// TwinCAT 3 PLC project Untitled1
// ProgramVersion: 3.1.4024.0
// libraries:
//   Tc2_MC2, * (Beckhoff Automation GmbH)
//   Tc2_MC2_Drive, * (Beckhoff Automation GmbH)
//   Tc2_Standard, * (Beckhoff Automation GmbH)
//   Tc2_System, * (Beckhoff Automation GmbH)
//   Tc3_Module, * (Beckhoff Automation GmbH)
// project tree:
//   GVLs/ GVL.TcGVL
//   / PlcTask.TcTTO
//   POUs/ Get_PID_Gain.TcPOU, Init.TcPOU, MAIN.TcPOU
// real-time tasks:
//   TASK PlcTask: cycle T#10ms, priority 20, ADS port 350
// motion (NC):
//   TASK NC-Task 1 SAF: cycle T#2ms, priority 4, ADS port 501
//   TASK NC-Task 1 SVB: cycle T#10ms, priority 8, ADS port 511
//   AXIS Axis 1 (id 1)
//     OtherSettings: AllowMotionCmdToSlave=true
//     encoder EncType=19
//       EncPara: MaxCount=#xffffffff
//     drive DrvType=16
//       DrvPara: MaxCount=#xffffffff, DriveControlDWord=#x00020100
//         Analog: TorqueSetpointScale=10, ScaleFactorActTorque=0.1
//         TimeComp: TaskDelayCycles=1
//     controller CtrType=1
//       CtrPara: PriorControlFactor=1
//         PosDiffControl: Enable=false
//         Observer: BandWidth=20
//   AXIS Axis 2 (id 2)
//     OtherSettings: AllowMotionCmdToSlave=true
//     encoder EncType=19
//       EncPara: MaxCount=#xffffffff
//     drive DrvType=16
//       DrvPara: MaxCount=#xffffffff, DriveControlDWord=#x00020100
//         Analog: TorqueSetpointScale=10, ScaleFactorActTorque=0.1
//         TimeComp: TaskDelayCycles=1
//     controller CtrType=1
//       CtrPara: PriorControlFactor=1
//         PosDiffControl: Enable=false
//         Observer: BandWidth=20
// I/O:
//   DEVICE Device 3 (EtherCAT), AmsNetId 169.254.80.96.4.1
//     Drive 1 (MADHT1505BA1) [MADHT1505BA1]
//     Drive 2 (MADHT1507BA1) [MADHT1507BA1]
// variable links:
//   NC-Task 1 SAF/Axes/Axis 1 <-> Device 3 (EtherCAT)/Drive 1 (MADHT1505BA1)
//     Drive/Inputs/In/nDataIn1 <-> Transmit PDO mapping 1/Following error actual value
//     Drive/Inputs/In/nState1 <-> Transmit PDO mapping 1/Statusword
//     Drive/Inputs/In/nState2 <-> Transmit PDO mapping 1/Statusword @bit 8
//     Drive/Inputs/In/nState4 @bit 1 <-> WcState/InputToggle
//     Drive/Inputs/In/nState4 <-> WcState/WcState
//     Drive/Inputs/In/nState5 <-> Transmit PDO mapping 1/Modes of operation display
//     Drive/Outputs/Out/nCtrl1 <-> Receive PDO mapping 1/Controlword
//     Drive/Outputs/Out/nCtrl2 <-> Receive PDO mapping 1/Controlword @bit 8
//     Drive/Outputs/Out/nCtrl5 <-> Receive PDO mapping 1/Modes of operation
//     Drive/Outputs/Out/nDataOut1 <-> Receive PDO mapping 1/Target position
//     Enc/Inputs/In/nDataIn1 <-> Transmit PDO mapping 1/Position actual value
//     Enc/Inputs/In/nDataIn3 <-> Transmit PDO mapping 1/Touch probe pos1 pos value
//     Enc/Inputs/In/nState4 @bit 1 <-> WcState/InputToggle
//     Enc/Inputs/In/nState4 <-> WcState/WcState
//     Enc/Inputs/In/nState5 <-> Transmit PDO mapping 1/Touch probe status
//     Enc/Inputs/In/nState6 <-> Transmit PDO mapping 1/Touch probe status @bit 8
//     Enc/Outputs/Out/nCtrl5 <-> Receive PDO mapping 1/Touch probe function
//     Enc/Outputs/Out/nCtrl6 <-> Receive PDO mapping 1/Touch probe function @bit 8
//   NC-Task 1 SAF/Axes/Axis 2 <-> Device 3 (EtherCAT)/Drive 2 (MADHT1507BA1)
//     Drive/Inputs/In/nDataIn1 <-> Transmit PDO mapping 1/Following error actual value
//     Drive/Inputs/In/nState1 <-> Transmit PDO mapping 1/Statusword
//     Drive/Inputs/In/nState2 <-> Transmit PDO mapping 1/Statusword @bit 8
//     Drive/Inputs/In/nState4 @bit 1 <-> WcState/InputToggle
//     Drive/Inputs/In/nState4 <-> WcState/WcState
//     Drive/Inputs/In/nState5 <-> Transmit PDO mapping 1/Modes of operation display
//     Drive/Outputs/Out/nCtrl1 <-> Receive PDO mapping 1/Controlword
//     Drive/Outputs/Out/nCtrl2 <-> Receive PDO mapping 1/Controlword @bit 8
//     Drive/Outputs/Out/nCtrl5 <-> Receive PDO mapping 1/Modes of operation
//     Drive/Outputs/Out/nDataOut1 <-> Receive PDO mapping 1/Target position
//     Enc/Inputs/In/nDataIn1 <-> Transmit PDO mapping 1/Position actual value
//     Enc/Inputs/In/nDataIn3 <-> Transmit PDO mapping 1/Touch probe pos1 pos value
//     Enc/Inputs/In/nState4 @bit 1 <-> WcState/InputToggle
//     Enc/Inputs/In/nState4 <-> WcState/WcState
//     Enc/Inputs/In/nState5 <-> Transmit PDO mapping 1/Touch probe status
//     Enc/Inputs/In/nState6 <-> Transmit PDO mapping 1/Touch probe status @bit 8
//     Enc/Outputs/Out/nCtrl5 <-> Receive PDO mapping 1/Touch probe function
//     Enc/Outputs/Out/nCtrl6 <-> Receive PDO mapping 1/Touch probe function @bit 8
//   Untitled1/Untitled1 Instance <-> NC-Task 1 SAF/Axes/Axis 1
//     PlcTask Inputs/GVL.AxisY.NcToPlc <-> Outputs/ToPlc
//     PlcTask Outputs/GVL.AxisY.PlcToNc <-> Inputs/FromPlc
//   Untitled1/Untitled1 Instance <-> NC-Task 1 SAF/Axes/Axis 2
//     PlcTask Inputs/GVL.AxisX.NcToPlc <-> Outputs/ToPlc
//     PlcTask Outputs/GVL.AxisX.PlcToNc <-> Inputs/FromPlc

CONFIGURATION Untitled1
    RESOURCE PLC ON TwinCAT3
        TASK PlcTask(INTERVAL := T#10ms, PRIORITY := 20);
        PROGRAM MAIN WITH PlcTask : MAIN;
    END_RESOURCE
END_CONFIGURATION

// ---- GVLs/GVL.TcGVL
{attribute 'qualified_only'}
VAR_GLOBAL
			AxisX : AXIS_REF;
			AxisY : AXIS_REF;
			
			//Moter Power	
			AxisX_Power_Fuc : MC_Power;
			AxisY_Power_Fuc : MC_Power;
					
			OnMoterX : BOOL;
			OnMoterY : BOOL;
			
			//***************Stop***********//
			X_Stop : MC_Stop;
			X_Stop_EX :BOOL :=FALSE;
			Y_Stop : MC_Stop;
			Y_Stop_EX :BOOL :=FALSE;
			//**************Jog***********//
			
			X_Jog : MC_Jog;
			Y_Jog : MC_Jog;
			X_FW : BOOL :=FALSE;
			X_BW : BOOL :=FALSE;
			//**************Pos_Offset_Clear***********//
			
			X_Pos_Offset_EX  : BOOL :=FALSE;
			Y_Pos_Offset_EX : BOOL :=FALSE;
			
			
			//***************Moter Move***************//
			AxisX_AbMove_Fuc :MC_MoveAbsolute;
			AxisY_AbMove_Fuc :MC_MoveAbsolute;
			
			//Moter GetVelocity
			X_GetVel: MC_ReadActualVelocity;
   			Y_GetVel: MC_ReadActualVelocity;
			X_Vel  : LREAL;
			Y_Vel  : LREAL;	
			
			//Moter GetPosition
			X_GetPos :MC_ReadActualPosition;
			Y_GetPos :MC_ReadActualPosition;
	  		X_Pos : LREAL;	  	  
	  		Y_Pos : LREAL;
			
			//Input
			X_Command_Vel : LREAL := 200;     
			X_Command_Acc : LREAL :=200;
			X_Command_Dec : LREAL :=200;
			X_AbMove_Ex : BOOL := FALSE;
			X_Command_Pos : LREAL :=0;
			
			Y_Command_Vel : LREAL := 200;     
			Y_Command_Acc : LREAL := 200;
			Y_Command_Dec : LREAL := 200;
			Y_AbMove_Ex : BOOL := FALSE;
			Y_Command_Pos : LREAL := 0;
			
				
			//Output
			X_Busy : BOOL;
			Y_Busy : BOOL;
			
			X_Error :BOOL;
			Y_Error :BOOL;
			
			X_ErrorID :UDINT;
			Y_ErrorID :UDINT;
			
			X_Done : BOOL;
			Y_Done : BOOL;	
		 //***************Moter Move End***************//
			
		//PID 
			
       		 fbCoEReadP_X:FB_CoERead;
			fbCoEReadI_X:FB_CoERead;
			fbCoEReadD_X:FB_CoERead;
			
			fbCoEReadP_Y:FB_CoERead;
			fbCoEReadI_Y:FB_CoERead;
			fbCoEReadD_Y:FB_CoERead;
			
			fbCoERead_Y:FB_CoERead;
			
			Index: WORD :=16#3100; 
			X_Gain: WORD :=400 ;
			Y_Gain: WORD :=400 ;
			X_COE_Ex :BOOL :=FALSE;
			Y_COE_Ex :BOOL :=FALSE;
			CompleteAccess: BOOL := FALSE; 
   			Success: BOOL; 
			
			X_GetP_Gain : WORD;
			X_GetI_Gain : WORD;
			X_GetD_Gain : WORD;
			X_CoERead_EX  :BOOL:=TRUE;
			
			Y_GetP_Gain : WORD;
			Y_GetI_Gain : WORD;
			Y_GetD_Gain : WORD;
			Y_CoERead_EX  :BOOL:=TRUE;
			//PID End
END_VAR

// ---- POUs/MAIN.TcPOU
PROGRAM MAIN
VAR
		Y_SetZero_Func: MC_SetPosition;
	
	    X_SetZero_Func: MC_SetPosition;
END_VAR


Y_SetZero_Func.Options.ClearPositionOffset :=TRUE;
Y_SetZero_Func(
		Axis :=GVL.AxisX,
		Position := ,
		Execute := GVL.X_Pos_Offset_EX,
);

X_SetZero_Func.Options.ClearPositionOffset :=TRUE;
X_SetZero_Func(
		Axis :=GVL.AxisY,
		Position := ,
		Execute := GVL.Y_Pos_Offset_EX,
);


Init();
Get_PID_Gain();


GVL.AxisX_Power_Fuc.Enable := GVL.OnMoterX;
GVL.AxisY_Power_Fuc.Enable := GVL.OnMoterY;



GVL.AxisX_AbMove_Fuc.Execute := GVL.X_AbMove_Ex;

IF NOT GVL.X_Busy THEN	
	GVL.X_AbMove_Ex := FALSE;
END_IF



GVL.AxisY_AbMove_Fuc.Execute := GVL.Y_AbMove_Ex;
IF NOT GVL.Y_Busy THEN	
	GVL.Y_AbMove_Ex := FALSE;
END_IF

END_PROGRAM

// ---- POUs/Init.TcPOU
FUNCTION Init : BOOL
VAR_INPUT
END_VAR
VAR
	IsComplete : BOOL;
END_VAR


GVL.X_Stop(
	 Axis := GVL.AxisX,
	 Execute :=GVL.X_Stop_EX
);

GVL.Y_Stop(
	 Axis := GVL.AxisY,
	 Execute :=GVL.Y_Stop_EX
);

GVL.X_Jog(

    Axis := GVL.AxisX,

    JogForward := GVL.X_FW,

    JogBackwards := GVL.X_BW,

    Position := 50,

    Velocity := 500,

    Mode := E_JogMode.MC_JOGMODE_INCHING
);



GVL.AxisX_Power_Fuc(
			Axis := GVL.AxisX,
			Enable_Negative :=TRUE,
			Enable_Positive := TRUE,
			Override := 100,
			Enable :=GVL.OnMoterX
			);	
			
GVL.AxisY_Power_Fuc(
			Axis := GVL.AxisY,
			Enable_Negative :=TRUE,
			Enable_Positive := TRUE,
			Override := 100,
			Enable :=GVL.OnMoterY
			);	
			
GVL.AxisX_AbMove_Fuc(
	Axis := GVL.AxisX,
	Acceleration := GVL.X_Command_Acc,
	Velocity := GVL.X_Command_Vel,
	Deceleration := GVL.X_Command_Dec,
	Position :=GVL.X_Command_Pos,
	Busy => GVL.X_Busy,
	Done => GVL.X_Done
	);
	
GVL.AxisY_AbMove_Fuc(
	Axis := GVL.AxisY,
	Acceleration := GVL.Y_Command_Acc,
	Velocity := GVL.Y_Command_Vel,
	Deceleration := GVL.Y_Command_Dec,
	Position :=GVL.Y_Command_Pos,
	Busy => GVL.Y_Busy,
	Error => GVL.Y_Error,
	ErrorID => GVL.Y_ErrorID,
	);
	
// Get Velocity and Position for PID Graph // 
GVL.X_GetVel(
	Axis :=GVL.AxisX,
	Enable := TRUE,
	ActualVelocity =>GVL.X_Vel
	);
GVL.Y_GetVel(
	Axis :=GVL.AxisY,
	Enable := TRUE,
	ActualVelocity =>GVL.Y_Vel
	);
GVL.X_GetPos(
	Axis := GVL.AxisX,
	Enable := TRUE,
	Position => GVL.X_Pos,
	);
GVL.Y_GetPos(
	Axis := GVL.AxisY,
	Enable := TRUE,
	Position => GVL.Y_Pos,
	);

END_FUNCTION

// ---- POUs/Get_PID_Gain.TcPOU
FUNCTION Get_PID_Gain : bool
VAR_INPUT
END_VAR
VAR
END_VAR

GVL.fbCoEReadP_X(
		Axis :=GVL.AxisX,		
		NetId := '169.254.80.96.1.1',   //target NetID 
  		Index := 16#3100,
  		pDstBuf := ADR(GVL.X_GetP_Gain), 
  		BufLen := SIZEOF(GVL.X_GetP_Gain), 
  		Execute := GVL.X_CoERead_EX, 
  		Timeout := T#1S, 	
	);	
GVL.fbCoEReadD_X(
		Axis :=GVL.AxisX,		
		NetId := '169.254.80.96.1.1', 
  		Index := 16#3101,
  		pDstBuf := ADR(GVL.X_GetD_Gain), 
  		BufLen := SIZEOF(GVL.X_GetD_Gain), 
  		Execute := GVL.X_CoERead_EX, 
  		Timeout := T#1S, 	
		
	);	
GVL.fbCoEReadI_X(
		Axis :=GVL.AxisX,		
		NetId := '169.254.80.96.1.1', 
  		Index := 16#3102,
  		pDstBuf := ADR(GVL.X_GetI_Gain), 
  		BufLen := SIZEOF(GVL.X_GetI_Gain), 
  		Execute := GVL.X_CoERead_EX, 
  		Timeout := T#1S, 	
	);	
GVL.X_CoERead_EX := FALSE;
	
GVL.fbCoEReadP_Y(
		Axis :=GVL.AxisY,		
		NetId := '169.254.80.96.1.1', 
  		Index := 16#3100,
  		pDstBuf := ADR(GVL.Y_GetP_Gain), 
  		BufLen := SIZEOF(GVL.Y_GetP_Gain), 
  		Execute := GVL.Y_CoERead_EX, 
  		Timeout := T#1S, 	
	);	
GVL.fbCoEReadD_Y(
		Axis :=GVL.AxisY,		
		NetId := '169.254.80.96.1.1', 
  		Index := 16#3101,
  		pDstBuf := ADR(GVL.Y_GetD_Gain), 
  		BufLen := SIZEOF(GVL.Y_GetD_Gain), 
  		Execute := GVL.Y_CoERead_EX, 
  		Timeout := T#1S, 	
		
	);	
GVL.fbCoEReadI_Y(
		Axis :=GVL.AxisY,		
		NetId := '169.254.80.96.1.1', 
  		Index := 16#3102,
  		pDstBuf := ADR(GVL.Y_GetI_Gain), 
  		BufLen := SIZEOF(GVL.X_GetI_Gain), 
  		Execute := GVL.Y_CoERead_EX, 
  		Timeout := T#1S, 	
	);	
GVL.Y_CoERead_EX := FALSE;

END_FUNCTION
